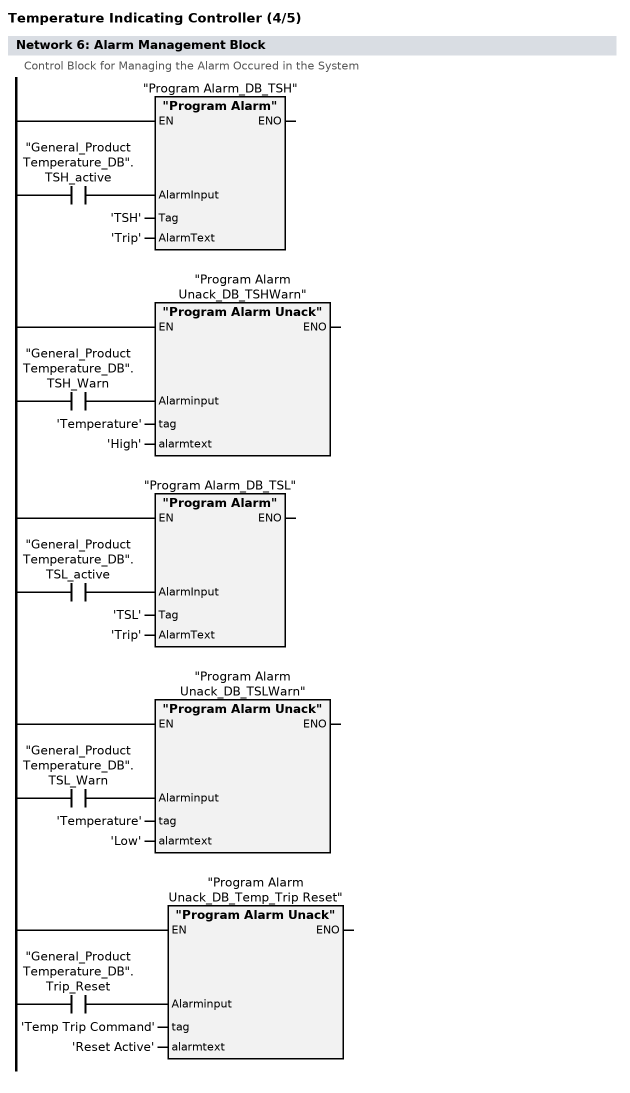
   RUNG wire#powerrail
      "Program Alarm_DB_TSH"(AlarmInput := wire#w1, Tag := 'TSH', AlarmText := 'Trip')
   END_RUNG
   RUNG wire#powerrail
      Contact( "General_Product Temperature_DB".TSH_active )
   END_RUNG wire#w1
   RUNG wire#powerrail
      "Program Alarm Unack_DB_TSHWarn"(Alarminput := wire#w2, tag := 'Temperature', alarmtext := 'High')
   END_RUNG
   RUNG wire#powerrail
      Contact( "General_Product Temperature_DB".TSH_Warn )
   END_RUNG wire#w2
   RUNG wire#powerrail
      "Program Alarm_DB_TSL"(AlarmInput := wire#w3, Tag := 'TSL', AlarmText := 'Trip')
   END_RUNG
   RUNG wire#powerrail
      Contact( "General_Product Temperature_DB".TSL_active )
   END_RUNG wire#w3
   RUNG wire#powerrail
      "Program Alarm Unack_DB_TSLWarn"(Alarminput := wire#w4, tag := 'Temperature', alarmtext := 'Low')
   END_RUNG
   RUNG wire#powerrail
      Contact( "General_Product Temperature_DB".TSL_Warn )
   END_RUNG wire#w4
   RUNG wire#powerrail
      "Program Alarm Unack_DB_Temp_Trip Reset"(Alarminput := wire#w5, tag := 'Temp Trip Command', alarmtext := 'Reset Active')
   END_RUNG
   RUNG wire#powerrail
      Contact( "General_Product Temperature_DB".Trip_Reset )
   END_RUNG wire#w5
   // the same network as SCL:
   "Program Alarm_DB_TSH"(AlarmInput := "General_Product Temperature_DB".TSH_active,   // "Program Alarm"
                          Tag := 'TSH',
                          AlarmText := 'Trip');
   "Program Alarm Unack_DB_TSHWarn"(Alarminput := "General_Product Temperature_DB".TSH_Warn,   // "Program Alarm Unack"
                           tag := 'Temperature',
                           alarmtext := 'High');
   "Program Alarm_DB_TSL"(AlarmInput := "General_Product Temperature_DB".TSL_active,   // "Program Alarm"
                          Tag := 'TSL',
                          AlarmText := 'Trip');
   "Program Alarm Unack_DB_TSLWarn"(Alarminput := "General_Product Temperature_DB".TSL_Warn,   // "Program Alarm Unack"
                           tag := 'Temperature',
                           alarmtext := 'Low');
   "Program Alarm Unack_DB_Temp_Trip Reset"(Alarminput := "General_Product Temperature_DB".Trip_Reset,   // "Program Alarm Unack"
                           tag := 'Temp Trip Command',
                           alarmtext := 'Reset Active');
END_REGION

REGION Network 7: User Additional Feature
   // Put additional feature that user can use to easier the system operation
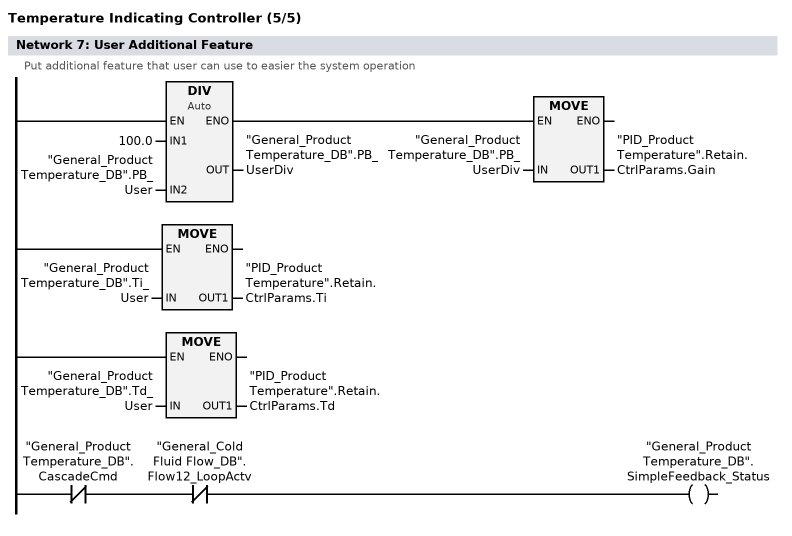
   RUNG wire#powerrail
      Div(in1 := 100.0, in2 := "General_Product Temperature_DB".PB_User, out => "General_Product Temperature_DB".PB_UserDiv)
      Move(in := "General_Product Temperature_DB".PB_UserDiv, out1 => "PID_Product Temperature".Retain.CtrlParams.Gain)
   END_RUNG
   RUNG wire#powerrail
      Move(in := "General_Product Temperature_DB".Ti_User, out1 => "PID_Product Temperature".Retain.CtrlParams.Ti)
   END_RUNG
   RUNG wire#powerrail
      Move(in := "General_Product Temperature_DB".Td_User, out1 => "PID_Product Temperature".Retain.CtrlParams.Td)
   END_RUNG
   RUNG wire#powerrail
      I_Contact( "General_Product Temperature_DB".CascadeCmd )
      I_Contact( "General_Cold Fluid Flow_DB".Flow12_LoopActv )
      Coil( "General_Product Temperature_DB".SimpleFeedback_Status )
   END_RUNG
   // the same network as SCL:
   "General_Product Temperature_DB".PB_UserDiv := 100.0 / "General_Product Temperature_DB".PB_User;
   "PID_Product Temperature".Retain.CtrlParams.Gain := "General_Product Temperature_DB".PB_UserDiv;
   "PID_Product Temperature".Retain.CtrlParams.Ti := "General_Product Temperature_DB".Ti_User;
   "PID_Product Temperature".Retain.CtrlParams.Td := "General_Product Temperature_DB".Td_User;
   "General_Product Temperature_DB".SimpleFeedback_Status := NOT "General_Product Temperature_DB".CascadeCmd AND NOT "General_Cold Fluid Flow_DB".Flow12_LoopActv;
END_REGION
END_ORGANIZATION_BLOCK

ORGANIZATION_BLOCK "Flow Indicating Controller 11"   // OB33, LAD, CyclicInterrupt
TITLE = Flow Indicator Controller 11 (Hot Fluid)
{ S7_Optimized_Access := 'TRUE' }
VERSION : 0.1
// Ladder and Block Program to control flowrate of Hot Fluid (Tank Input)
   VAR_INPUT
      Initial_Call : Bool;   // Initial call of this OB
      Event_Count : Int;   // Events discarded
   END_VAR
BEGIN

REGION Network 1: User Setpoint
   // User input their Setpoint for flowrate in L/s  converted into Real Number for PID Setpoint (0-100)
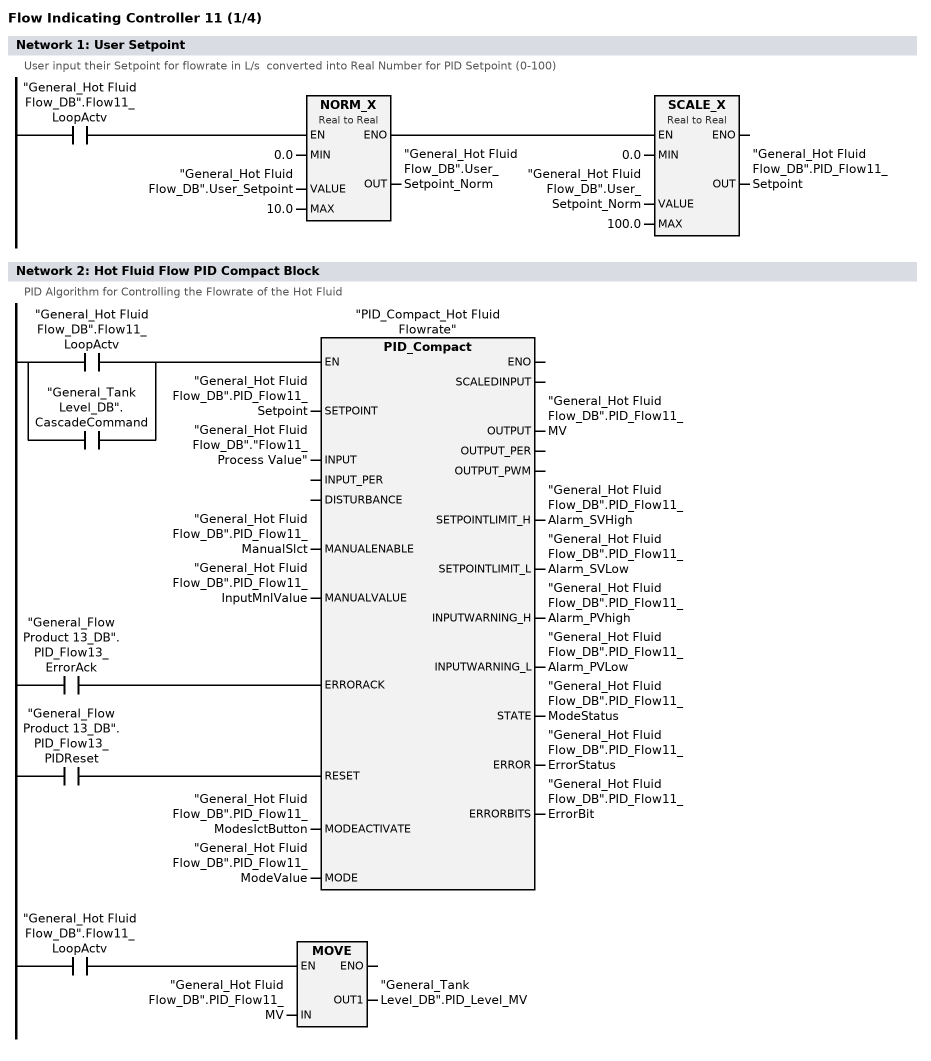
   RUNG wire#powerrail
      Contact( "General_Hot Fluid Flow_DB".Flow11_LoopActv )
      { S7_Templates := "[SrcType := Real, DestType := Real]" } Normalize(min := 0.0, value := "General_Hot Fluid Flow_DB".User_Setpoint, max := 10.0, out => "General_Hot Fluid Flow_DB".User_Setpoint_Norm)
      { S7_Templates := "[SrcType := Real, DestType := Real]" } Scale(min := 0.0, value := "General_Hot Fluid Flow_DB".User_Setpoint_Norm, max := 100.0, out => "General_Hot Fluid Flow_DB".PID_Flow11_Setpoint)
   END_RUNG
   // the same network as SCL:
   IF "General_Hot Fluid Flow_DB".Flow11_LoopActv THEN
       "General_Hot Fluid Flow_DB".User_Setpoint_Norm := NORM_X(MIN := 0.0, VALUE := "General_Hot Fluid Flow_DB".User_Setpoint, MAX := 10.0);
       "General_Hot Fluid Flow_DB".PID_Flow11_Setpoint := SCALE_X(MIN := 0.0, VALUE := "General_Hot Fluid Flow_DB".User_Setpoint_Norm, MAX := 100.0);
   END_IF;
END_REGION

REGION Network 2: Hot Fluid Flow PID Compact Block
   // PID Algorithm for Controlling the Flowrate of the Hot Fluid
   IF "General_Hot Fluid Flow_DB".Flow11_LoopActv OR "General_Tank Level_DB".CascadeCommand THEN
       "PID_Compact_Hot Fluid Flowrate"(Setpoint := "General_Hot Fluid Flow_DB".PID_Flow11_Setpoint,   // PID_Compact
                               Input := "General_Hot Fluid Flow_DB"."Flow11_Process Value",
                               ManualEnable := "General_Hot Fluid Flow_DB".PID_Flow11_ManualSlct,
                               ManualValue := "General_Hot Fluid Flow_DB".PID_Flow11_InputMnlValue,
                               ErrorAck := "General_Flow Product 13_DB".PID_Flow13_ErrorAck,
                               Reset := "General_Flow Product 13_DB".PID_Flow13_PIDReset,
                               ModeActivate := "General_Hot Fluid Flow_DB".PID_Flow11_ModeslctButton,
                               Mode := "General_Hot Fluid Flow_DB".PID_Flow11_ModeValue,
                               Output => "General_Hot Fluid Flow_DB".PID_Flow11_MV,
                               SetpointLimit_H => "General_Hot Fluid Flow_DB".PID_Flow11_Alarm_SVHigh,
                               SetpointLimit_L => "General_Hot Fluid Flow_DB".PID_Flow11_Alarm_SVLow,
                               InputWarning_H => "General_Hot Fluid Flow_DB".PID_Flow11_Alarm_PVhigh,
                               InputWarning_L => "General_Hot Fluid Flow_DB".PID_Flow11_Alarm_PVLow,
                               State => "General_Hot Fluid Flow_DB".PID_Flow11_ModeStatus,
                               Error => "General_Hot Fluid Flow_DB".PID_Flow11_ErrorStatus,
                               ErrorBits => "General_Hot Fluid Flow_DB".PID_Flow11_ErrorBit);
   END_IF;
   IF "General_Hot Fluid Flow_DB".Flow11_LoopActv THEN
       "General_Tank Level_DB".PID_Level_MV := "General_Hot Fluid Flow_DB".PID_Flow11_MV;
   END_IF;
END_REGION

REGION Network 3: Hot Fluid Process Control Block
   // Process for Flowrate as First Order System
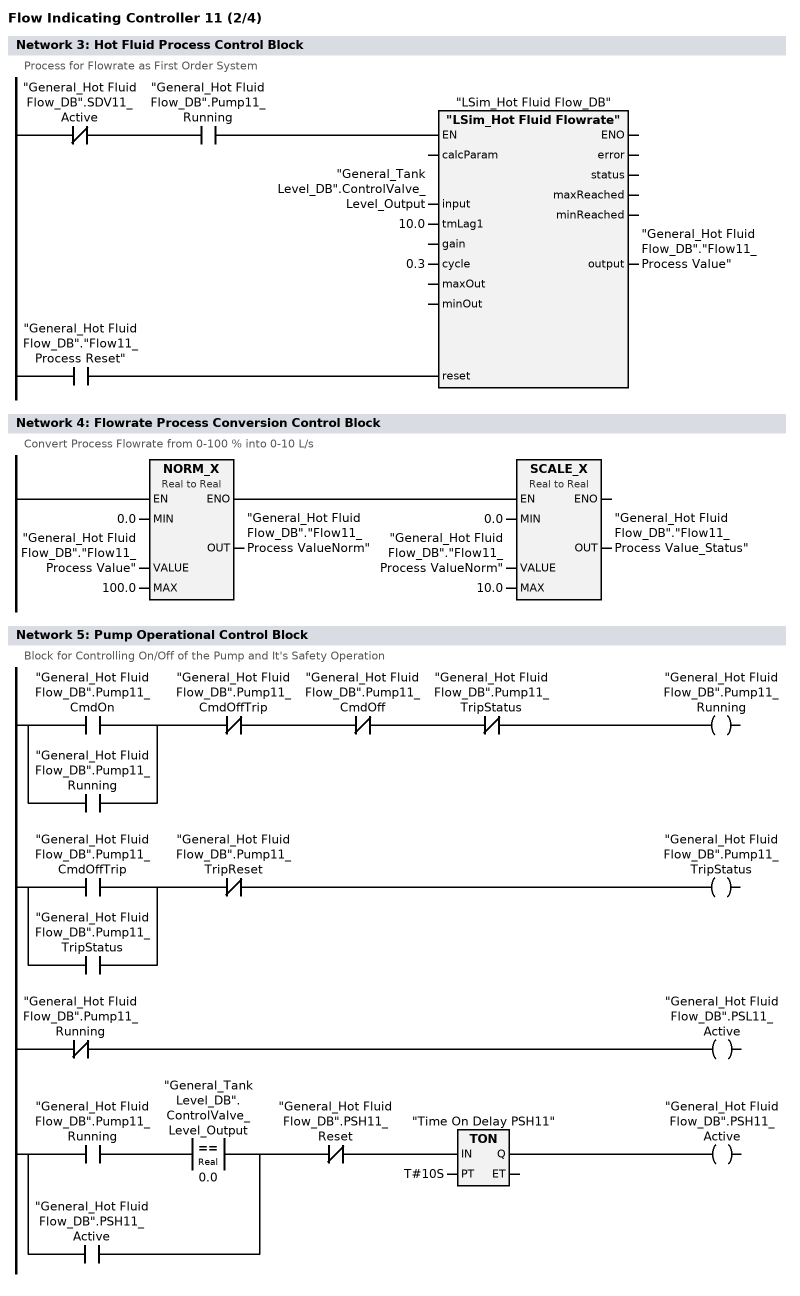
   RUNG wire#powerrail
      I_Contact( "General_Hot Fluid Flow_DB".SDV11_Active )
      Contact( "General_Hot Fluid Flow_DB".Pump11_Running )
      "LSim_Hot Fluid Flow_DB"(reset := wire#w1, calcParam :=, input := "General_Tank Level_DB".ControlValve_Level_Output, tmLag1 := 10.0, gain :=, cycle := 0.3, maxOut :=, minOut :=, error =>, status =>, maxReached =>, minReached =>, output => "General_Hot Fluid Flow_DB"."Flow11_Process Value")
   END_RUNG
   RUNG wire#powerrail
      Contact( "General_Hot Fluid Flow_DB"."Flow11_Process Reset" )
   END_RUNG wire#w1
   // the same network as SCL:
   IF NOT "General_Hot Fluid Flow_DB".SDV11_Active AND "General_Hot Fluid Flow_DB".Pump11_Running THEN
       "LSim_Hot Fluid Flow_DB"(input := "General_Tank Level_DB".ControlValve_Level_Output,   // "LSim_Hot Fluid Flowrate"
                               tmLag1 := 10.0,
                               cycle := 0.3,
                               reset := "General_Hot Fluid Flow_DB"."Flow11_Process Reset",
                               output => "General_Hot Fluid Flow_DB"."Flow11_Process Value");
   END_IF;
END_REGION

REGION Network 4: Flowrate Process Conversion Control Block
   // Convert Process Flowrate from 0-100 % into 0-10 L/s
   RUNG wire#powerrail
      { S7_Templates := "[SrcType := Real, DestType := Real]" } Normalize(min := 0.0, value := "General_Hot Fluid Flow_DB"."Flow11_Process Value", max := 100.0, out => "General_Hot Fluid Flow_DB"."Flow11_Process ValueNorm")
      { S7_Templates := "[SrcType := Real, DestType := Real]" } Scale(min := 0.0, value := "General_Hot Fluid Flow_DB"."Flow11_Process ValueNorm", max := 10.0, out => "General_Hot Fluid Flow_DB"."Flow11_Process Value_Status")
   END_RUNG
   // the same network as SCL:
   "General_Hot Fluid Flow_DB"."Flow11_Process ValueNorm" := NORM_X(MIN := 0.0, VALUE := "General_Hot Fluid Flow_DB"."Flow11_Process Value", MAX := 100.0);
   "General_Hot Fluid Flow_DB"."Flow11_Process Value_Status" := SCALE_X(MIN := 0.0, VALUE := "General_Hot Fluid Flow_DB"."Flow11_Process ValueNorm", MAX := 10.0);
END_REGION

REGION Network 5: Pump Operational Control Block
   // Block for Controlling On/Off of the Pump and It's Safety Operation
   "General_Hot Fluid Flow_DB".Pump11_Running := ("General_Hot Fluid Flow_DB".Pump11_CmdOn OR "General_Hot Fluid Flow_DB".Pump11_Running) AND NOT "General_Hot Fluid Flow_DB".Pump11_CmdOffTrip AND NOT "General_Hot Fluid Flow_DB".Pump11_CmdOff AND NOT "General_Hot Fluid Flow_DB".Pump11_TripStatus;
   "General_Hot Fluid Flow_DB".Pump11_TripStatus := ("General_Hot Fluid Flow_DB".Pump11_CmdOffTrip OR "General_Hot Fluid Flow_DB".Pump11_TripStatus) AND NOT "General_Hot Fluid Flow_DB".Pump11_TripReset;
   "General_Hot Fluid Flow_DB".PSL11_Active := NOT "General_Hot Fluid Flow_DB".Pump11_Running;
   "Time On Delay PSH11".TON(IN := (("General_Hot Fluid Flow_DB".Pump11_Running AND ("General_Tank Level_DB".ControlValve_Level_Output = 0.0)) OR "General_Hot Fluid Flow_DB".PSH11_Active) AND NOT "General_Hot Fluid Flow_DB".PSH11_Reset,
                           PT := T#10S);
   "General_Hot Fluid Flow_DB".PSH11_Active := "Time On Delay PSH11".Q;
END_REGION

REGION Network 6: Alarm Management Block
   // Control Block for Managing the Alarm Occured in the System
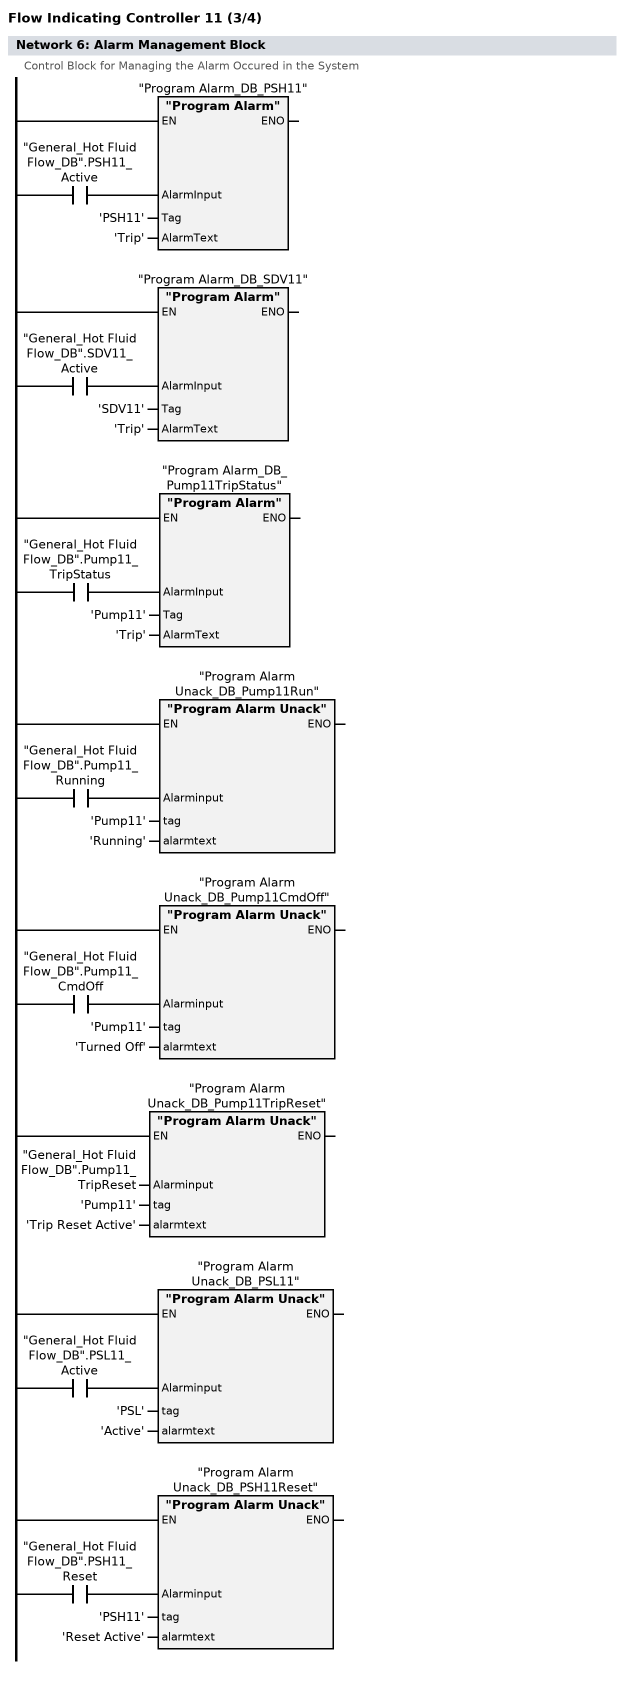
   RUNG wire#powerrail
      "Program Alarm_DB_PSH11"(AlarmInput := wire#w1, Tag := 'PSH11', AlarmText := 'Trip')
   END_RUNG
   RUNG wire#powerrail
      Contact( "General_Hot Fluid Flow_DB".PSH11_Active )
   END_RUNG wire#w1
   RUNG wire#powerrail
      "Program Alarm_DB_SDV11"(AlarmInput := wire#w2, Tag := 'SDV11', AlarmText := 'Trip')
   END_RUNG
   RUNG wire#powerrail
      Contact( "General_Hot Fluid Flow_DB".SDV11_Active )
   END_RUNG wire#w2
   RUNG wire#powerrail
      "Program Alarm_DB_Pump11TripStatus"(AlarmInput := wire#w3, Tag := 'Pump11', AlarmText := 'Trip')
   END_RUNG
   RUNG wire#powerrail
      Contact( "General_Hot Fluid Flow_DB".Pump11_TripStatus )
   END_RUNG wire#w3
   RUNG wire#powerrail
      "Program Alarm Unack_DB_Pump11Run"(Alarminput := wire#w4, tag := 'Pump11', alarmtext := 'Running')
   END_RUNG
   RUNG wire#powerrail
      Contact( "General_Hot Fluid Flow_DB".Pump11_Running )
   END_RUNG wire#w4
   RUNG wire#powerrail
      "Program Alarm Unack_DB_Pump11CmdOff"(Alarminput := wire#w5, tag := 'Pump11', alarmtext := 'Turned Off')
   END_RUNG
   RUNG wire#powerrail
      Contact( "General_Hot Fluid Flow_DB".Pump11_CmdOff )
   END_RUNG wire#w5
   RUNG wire#powerrail
      "Program Alarm Unack_DB_Pump11TripReset"(Alarminput := "General_Hot Fluid Flow_DB".Pump11_TripReset, tag := 'Pump11', alarmtext := 'Trip Reset Active')
   END_RUNG
   RUNG wire#powerrail
      "Program Alarm Unack_DB_PSL11"(Alarminput := wire#w6, tag := 'PSL', alarmtext := 'Active')
   END_RUNG
   RUNG wire#powerrail
      Contact( "General_Hot Fluid Flow_DB".PSL11_Active )
   END_RUNG wire#w6
   RUNG wire#powerrail
      "Program Alarm Unack_DB_PSH11Reset"(Alarminput := wire#w7, tag := 'PSH11', alarmtext := 'Reset Active')
   END_RUNG
   RUNG wire#powerrail
      Contact( "General_Hot Fluid Flow_DB".PSH11_Reset )
   END_RUNG wire#w7
   // the same network as SCL:
   "Program Alarm_DB_PSH11"(AlarmInput := "General_Hot Fluid Flow_DB".PSH11_Active,   // "Program Alarm"
                           Tag := 'PSH11',
                           AlarmText := 'Trip');
   "Program Alarm_DB_SDV11"(AlarmInput := "General_Hot Fluid Flow_DB".SDV11_Active,   // "Program Alarm"
                           Tag := 'SDV11',
                           AlarmText := 'Trip');
   "Program Alarm_DB_Pump11TripStatus"(AlarmInput := "General_Hot Fluid Flow_DB".Pump11_TripStatus,   // "Program Alarm"
                           Tag := 'Pump11',
                           AlarmText := 'Trip');
   "Program Alarm Unack_DB_Pump11Run"(Alarminput := "General_Hot Fluid Flow_DB".Pump11_Running,   // "Program Alarm Unack"
                           tag := 'Pump11',
                           alarmtext := 'Running');
   "Program Alarm Unack_DB_Pump11CmdOff"(Alarminput := "General_Hot Fluid Flow_DB".Pump11_CmdOff,   // "Program Alarm Unack"
                           tag := 'Pump11',
                           alarmtext := 'Turned Off');
   "Program Alarm Unack_DB_Pump11TripReset"(Alarminput := "General_Hot Fluid Flow_DB".Pump11_TripReset,   // "Program Alarm Unack"
                           tag := 'Pump11',
                           alarmtext := 'Trip Reset Active');
   "Program Alarm Unack_DB_PSL11"(Alarminput := "General_Hot Fluid Flow_DB".PSL11_Active,   // "Program Alarm Unack"
                           tag := 'PSL',
                           alarmtext := 'Active');
   "Program Alarm Unack_DB_PSH11Reset"(Alarminput := "General_Hot Fluid Flow_DB".PSH11_Reset,   // "Program Alarm Unack"
                           tag := 'PSH11',
                           alarmtext := 'Reset Active');
END_REGION

REGION Network 7: User Additional Feature
   // Put additional feature that user can use to easier the system operation
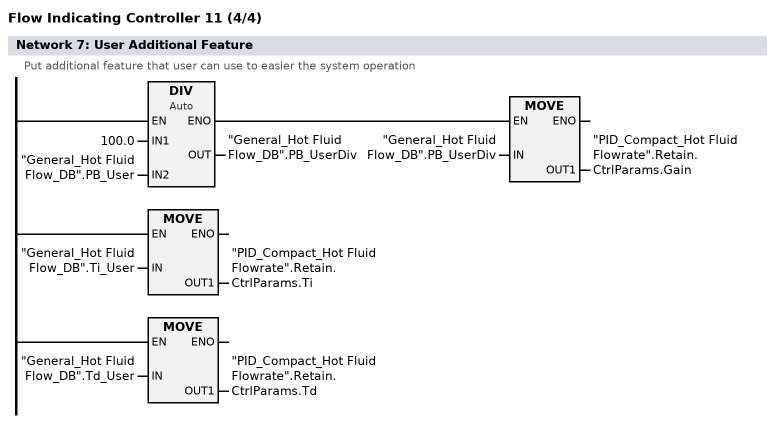
   RUNG wire#powerrail
      Div(in1 := 100.0, in2 := "General_Hot Fluid Flow_DB".PB_User, out => "General_Hot Fluid Flow_DB".PB_UserDiv)
      Move(in := "General_Hot Fluid Flow_DB".PB_UserDiv, out1 => "PID_Compact_Hot Fluid Flowrate".Retain.CtrlParams.Gain)
   END_RUNG
   RUNG wire#powerrail
      Move(in := "General_Hot Fluid Flow_DB".Ti_User, out1 => "PID_Compact_Hot Fluid Flowrate".Retain.CtrlParams.Ti)
   END_RUNG
   RUNG wire#powerrail
      Move(in := "General_Hot Fluid Flow_DB".Td_User, out1 => "PID_Compact_Hot Fluid Flowrate".Retain.CtrlParams.Td)
   END_RUNG
   // the same network as SCL:
   "General_Hot Fluid Flow_DB".PB_UserDiv := 100.0 / "General_Hot Fluid Flow_DB".PB_User;
   "PID_Compact_Hot Fluid Flowrate".Retain.CtrlParams.Gain := "General_Hot Fluid Flow_DB".PB_UserDiv;
   "PID_Compact_Hot Fluid Flowrate".Retain.CtrlParams.Ti := "General_Hot Fluid Flow_DB".Ti_User;
   "PID_Compact_Hot Fluid Flowrate".Retain.CtrlParams.Td := "General_Hot Fluid Flow_DB".Td_User;
END_REGION
END_ORGANIZATION_BLOCK

ORGANIZATION_BLOCK "Flow Indicating Controller 12"   // OB34, LAD, CyclicInterrupt
TITLE = Flow Indicator Controller 12 (Cold Fluid)
{ S7_Optimized_Access := 'TRUE' }
VERSION : 0.1
// Ladder and Block Program to control flowrate of Cold Fluid (Tank Input)
   VAR_INPUT
      Initial_Call : Bool;   // Initial call of this OB
      Event_Count : Int;   // Events discarded
   END_VAR
BEGIN

REGION Network 1: User Setpoint
   // User input their Setpoint for flowrate in L/s  converted into Real Number for PID Setpoint (0-100)
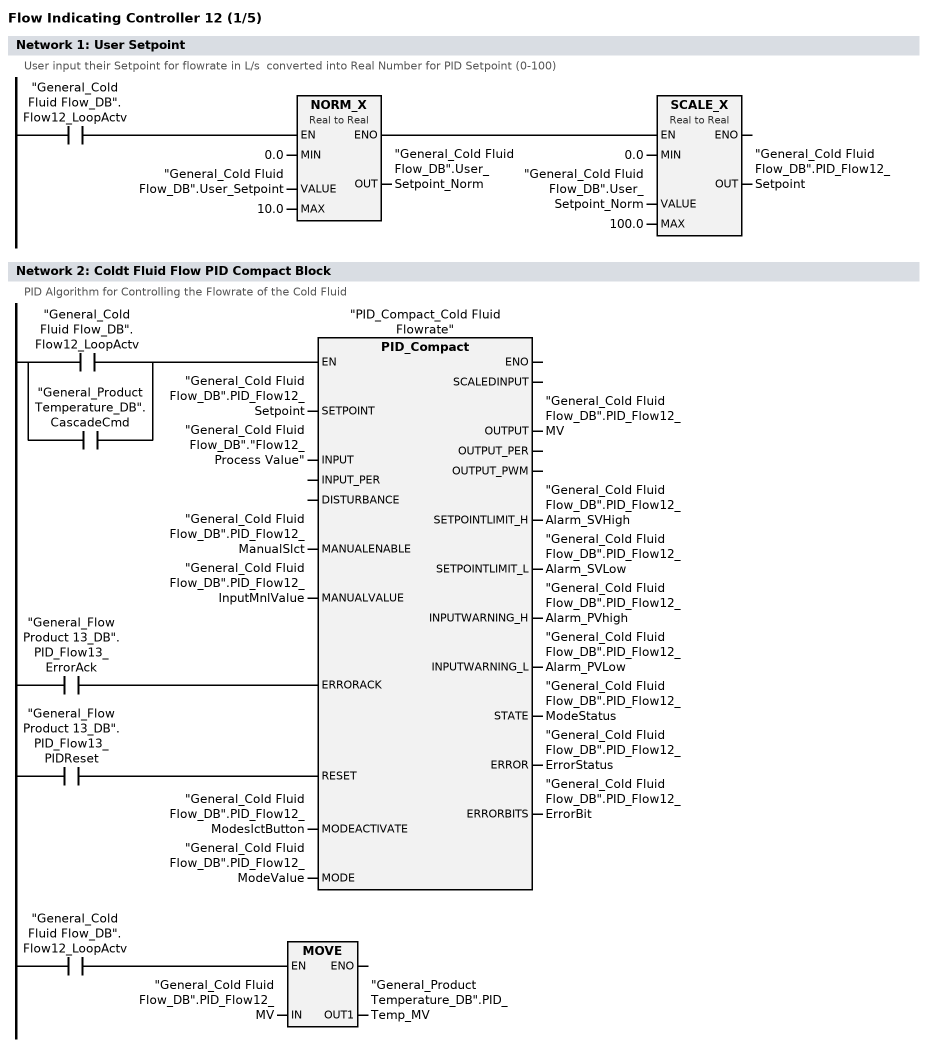
   RUNG wire#powerrail
      Contact( "General_Cold Fluid Flow_DB".Flow12_LoopActv )
      { S7_Templates := "[SrcType := Real, DestType := Real]" } Normalize(min := 0.0, value := "General_Cold Fluid Flow_DB".User_Setpoint, max := 10.0, out => "General_Cold Fluid Flow_DB".User_Setpoint_Norm)
      { S7_Templates := "[SrcType := Real, DestType := Real]" } Scale(min := 0.0, value := "General_Cold Fluid Flow_DB".User_Setpoint_Norm, max := 100.0, out => "General_Cold Fluid Flow_DB".PID_Flow12_Setpoint)
   END_RUNG
   // the same network as SCL:
   IF "General_Cold Fluid Flow_DB".Flow12_LoopActv THEN
       "General_Cold Fluid Flow_DB".User_Setpoint_Norm := NORM_X(MIN := 0.0, VALUE := "General_Cold Fluid Flow_DB".User_Setpoint, MAX := 10.0);
       "General_Cold Fluid Flow_DB".PID_Flow12_Setpoint := SCALE_X(MIN := 0.0, VALUE := "General_Cold Fluid Flow_DB".User_Setpoint_Norm, MAX := 100.0);
   END_IF;
END_REGION

REGION Network 2: Coldt Fluid Flow PID Compact Block
   // PID Algorithm for Controlling the Flowrate of the Cold Fluid
   IF "General_Cold Fluid Flow_DB".Flow12_LoopActv OR "General_Product Temperature_DB".CascadeCmd THEN
       "PID_Compact_Cold Fluid Flowrate"(Setpoint := "General_Cold Fluid Flow_DB".PID_Flow12_Setpoint,   // PID_Compact
                               Input := "General_Cold Fluid Flow_DB"."Flow12_Process Value",
                               ManualEnable := "General_Cold Fluid Flow_DB".PID_Flow12_ManualSlct,
                               ManualValue := "General_Cold Fluid Flow_DB".PID_Flow12_InputMnlValue,
                               ErrorAck := "General_Flow Product 13_DB".PID_Flow13_ErrorAck,
                               Reset := "General_Flow Product 13_DB".PID_Flow13_PIDReset,
                               ModeActivate := "General_Cold Fluid Flow_DB".PID_Flow12_ModeslctButton,
                               Mode := "General_Cold Fluid Flow_DB".PID_Flow12_ModeValue,
                               Output => "General_Cold Fluid Flow_DB".PID_Flow12_MV,
                               SetpointLimit_H => "General_Cold Fluid Flow_DB".PID_Flow12_Alarm_SVHigh,
                               SetpointLimit_L => "General_Cold Fluid Flow_DB".PID_Flow12_Alarm_SVLow,
                               InputWarning_H => "General_Cold Fluid Flow_DB".PID_Flow12_Alarm_PVhigh,
                               InputWarning_L => "General_Cold Fluid Flow_DB".PID_Flow12_Alarm_PVLow,
                               State => "General_Cold Fluid Flow_DB".PID_Flow12_ModeStatus,
                               Error => "General_Cold Fluid Flow_DB".PID_Flow12_ErrorStatus,
                               ErrorBits => "General_Cold Fluid Flow_DB".PID_Flow12_ErrorBit);
   END_IF;
   IF "General_Cold Fluid Flow_DB".Flow12_LoopActv THEN
       "General_Product Temperature_DB".PID_Temp_MV := "General_Cold Fluid Flow_DB".PID_Flow12_MV;
   END_IF;
END_REGION

REGION Network 3: Cold Fluid Process Control Block
   // Process for Flowrate as First Order System
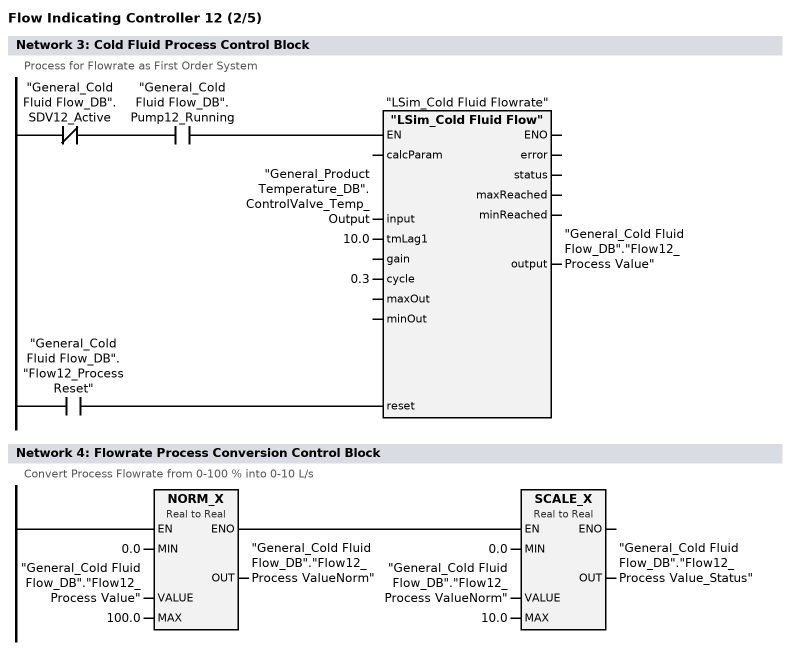
   RUNG wire#powerrail
      I_Contact( "General_Cold Fluid Flow_DB".SDV12_Active )
      Contact( "General_Cold Fluid Flow_DB".Pump12_Running )
      "LSim_Cold Fluid Flowrate"(reset := wire#w1, calcParam :=, input := "General_Product Temperature_DB".ControlValve_Temp_Output, tmLag1 := 10.0, gain :=, cycle := 0.3, maxOut :=, minOut :=, error =>, status =>, maxReached =>, minReached =>, output => "General_Cold Fluid Flow_DB"."Flow12_Process Value")
   END_RUNG
   RUNG wire#powerrail
      Contact( "General_Cold Fluid Flow_DB"."Flow12_Process Reset" )
   END_RUNG wire#w1
   // the same network as SCL:
   IF NOT "General_Cold Fluid Flow_DB".SDV12_Active AND "General_Cold Fluid Flow_DB".Pump12_Running THEN
       "LSim_Cold Fluid Flowrate"(input := "General_Product Temperature_DB".ControlValve_Temp_Output,   // "LSim_Cold Fluid Flow"
                               tmLag1 := 10.0,
                               cycle := 0.3,
                               reset := "General_Cold Fluid Flow_DB"."Flow12_Process Reset",
                               output => "General_Cold Fluid Flow_DB"."Flow12_Process Value");
   END_IF;
END_REGION

REGION Network 4: Flowrate Process Conversion Control Block
   // Convert Process Flowrate from 0-100 % into 0-10 L/s
   RUNG wire#powerrail
      { S7_Templates := "[SrcType := Real, DestType := Real]" } Normalize(min := 0.0, value := "General_Cold Fluid Flow_DB"."Flow12_Process Value", max := 100.0, out => "General_Cold Fluid Flow_DB"."Flow12_Process ValueNorm")
      { S7_Templates := "[SrcType := Real, DestType := Real]" } Scale(min := 0.0, value := "General_Cold Fluid Flow_DB"."Flow12_Process ValueNorm", max := 10.0, out => "General_Cold Fluid Flow_DB"."Flow12_Process Value_Status")
   END_RUNG
   // the same network as SCL:
   "General_Cold Fluid Flow_DB"."Flow12_Process ValueNorm" := NORM_X(MIN := 0.0, VALUE := "General_Cold Fluid Flow_DB"."Flow12_Process Value", MAX := 100.0);
   "General_Cold Fluid Flow_DB"."Flow12_Process Value_Status" := SCALE_X(MIN := 0.0, VALUE := "General_Cold Fluid Flow_DB"."Flow12_Process ValueNorm", MAX := 10.0);
END_REGION

REGION Network 5: Pump Operational Control Block
   // Block for Controlling On/Off of the Pump and It's Safety Operation
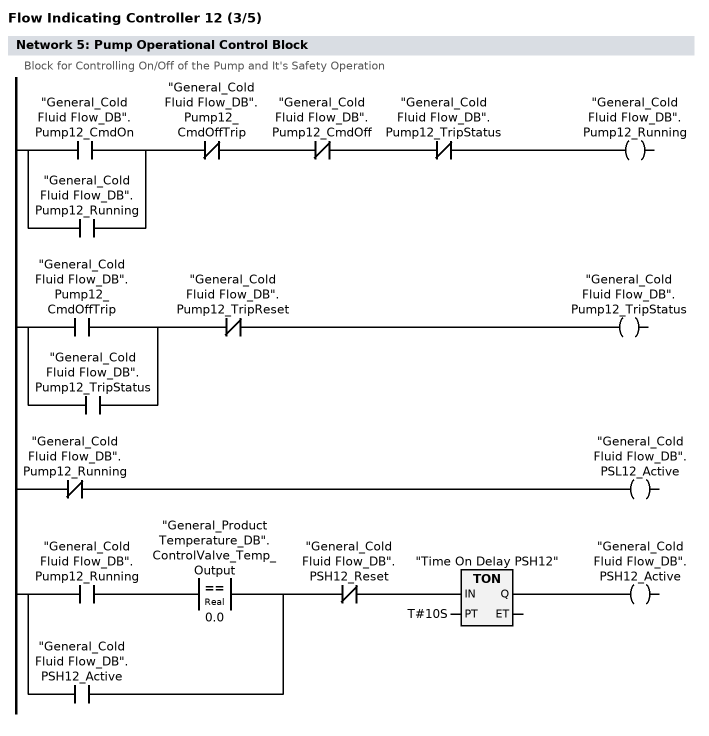
   "General_Cold Fluid Flow_DB".Pump12_Running := ("General_Cold Fluid Flow_DB".Pump12_CmdOn OR "General_Cold Fluid Flow_DB".Pump12_Running) AND NOT "General_Cold Fluid Flow_DB".Pump12_CmdOffTrip AND NOT "General_Cold Fluid Flow_DB".Pump12_CmdOff AND NOT "General_Cold Fluid Flow_DB".Pump12_TripStatus;
   "General_Cold Fluid Flow_DB".Pump12_TripStatus := ("General_Cold Fluid Flow_DB".Pump12_CmdOffTrip OR "General_Cold Fluid Flow_DB".Pump12_TripStatus) AND NOT "General_Cold Fluid Flow_DB".Pump12_TripReset;
   "General_Cold Fluid Flow_DB".PSL12_Active := NOT "General_Cold Fluid Flow_DB".Pump12_Running;
   "Time On Delay PSH12".TON(IN := (("General_Cold Fluid Flow_DB".Pump12_Running AND ("General_Product Temperature_DB".ControlValve_Temp_Output = 0.0)) OR "General_Cold Fluid Flow_DB".PSH12_Active) AND NOT "General_Cold Fluid Flow_DB".PSH12_Reset,
                           PT := T#10S);
   "General_Cold Fluid Flow_DB".PSH12_Active := "Time On Delay PSH12".Q;
END_REGION

REGION Network 6: Alarm Management Block
   // Control Block for Managing the Alarm Occured in the System
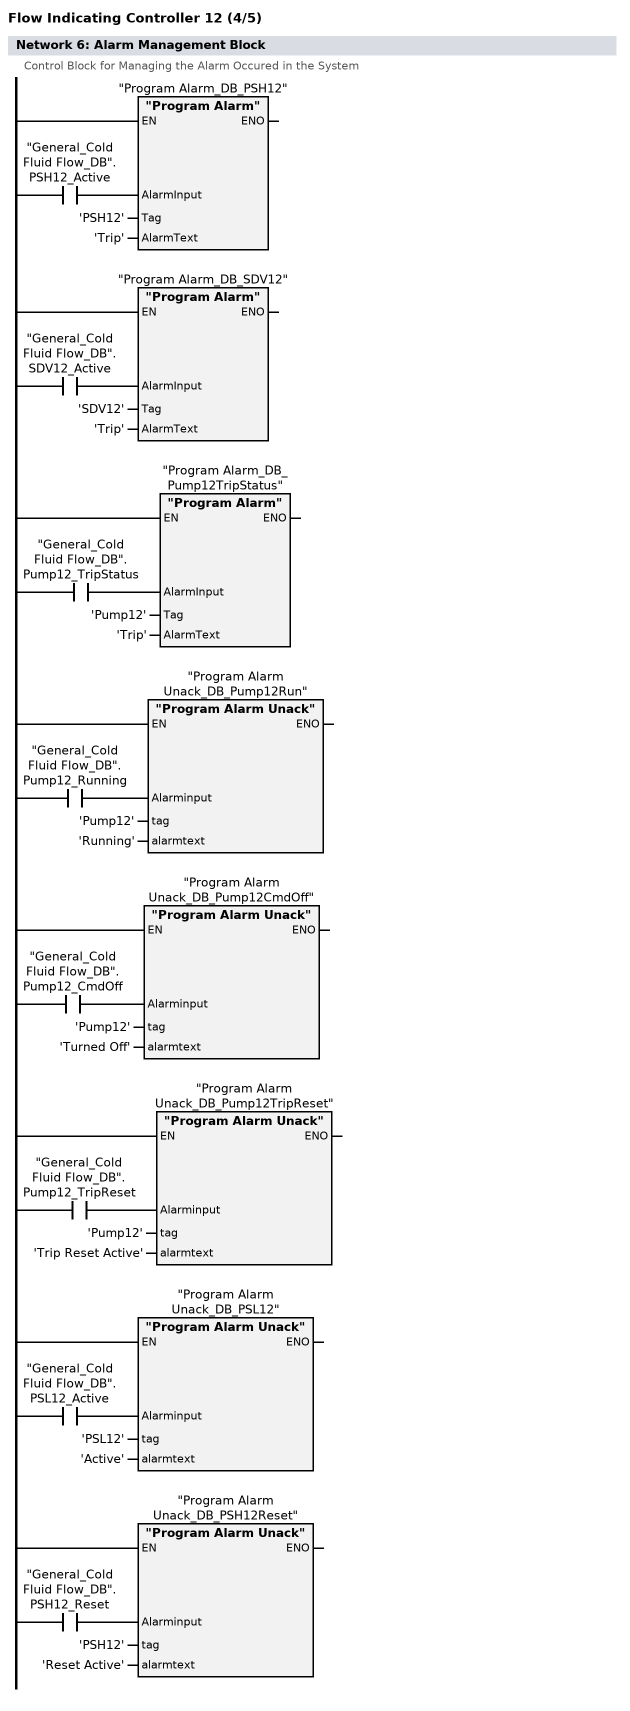
   RUNG wire#powerrail
      "Program Alarm_DB_PSH12"(AlarmInput := wire#w1, Tag := 'PSH12', AlarmText := 'Trip')
   END_RUNG
   RUNG wire#powerrail
      Contact( "General_Cold Fluid Flow_DB".PSH12_Active )
   END_RUNG wire#w1
   RUNG wire#powerrail
      "Program Alarm_DB_SDV12"(AlarmInput := wire#w2, Tag := 'SDV12', AlarmText := 'Trip')
   END_RUNG
   RUNG wire#powerrail
      Contact( "General_Cold Fluid Flow_DB".SDV12_Active )
   END_RUNG wire#w2
   RUNG wire#powerrail
      "Program Alarm_DB_Pump12TripStatus"(AlarmInput := wire#w3, Tag := 'Pump12', AlarmText := 'Trip')
   END_RUNG
   RUNG wire#powerrail
      Contact( "General_Cold Fluid Flow_DB".Pump12_TripStatus )
   END_RUNG wire#w3
   RUNG wire#powerrail
      "Program Alarm Unack_DB_Pump12Run"(Alarminput := wire#w4, tag := 'Pump12', alarmtext := 'Running')
   END_RUNG
   RUNG wire#powerrail
      Contact( "General_Cold Fluid Flow_DB".Pump12_Running )
   END_RUNG wire#w4
   RUNG wire#powerrail
      "Program Alarm Unack_DB_Pump12CmdOff"(Alarminput := wire#w5, tag := 'Pump12', alarmtext := 'Turned Off')
   END_RUNG
   RUNG wire#powerrail
      Contact( "General_Cold Fluid Flow_DB".Pump12_CmdOff )
   END_RUNG wire#w5
   RUNG wire#powerrail
      "Program Alarm Unack_DB_Pump12TripReset"(Alarminput := wire#w6, tag := 'Pump12', alarmtext := 'Trip Reset Active')
   END_RUNG
   RUNG wire#powerrail
      Contact( "General_Cold Fluid Flow_DB".Pump12_TripReset )
   END_RUNG wire#w6
   RUNG wire#powerrail
      "Program Alarm Unack_DB_PSL12"(Alarminput := wire#w7, tag := 'PSL12', alarmtext := 'Active')
   END_RUNG
   RUNG wire#powerrail
      Contact( "General_Cold Fluid Flow_DB".PSL12_Active )
   END_RUNG wire#w7
   RUNG wire#powerrail
      "Program Alarm Unack_DB_PSH12Reset"(Alarminput := wire#w8, tag := 'PSH12', alarmtext := 'Reset Active')
   END_RUNG
   RUNG wire#powerrail
      Contact( "General_Cold Fluid Flow_DB".PSH12_Reset )
   END_RUNG wire#w8
   // the same network as SCL:
   "Program Alarm_DB_PSH12"(AlarmInput := "General_Cold Fluid Flow_DB".PSH12_Active,   // "Program Alarm"
                           Tag := 'PSH12',
                           AlarmText := 'Trip');
   "Program Alarm_DB_SDV12"(AlarmInput := "General_Cold Fluid Flow_DB".SDV12_Active,   // "Program Alarm"
                           Tag := 'SDV12',
                           AlarmText := 'Trip');
   "Program Alarm_DB_Pump12TripStatus"(AlarmInput := "General_Cold Fluid Flow_DB".Pump12_TripStatus,   // "Program Alarm"
                           Tag := 'Pump12',
                           AlarmText := 'Trip');
   "Program Alarm Unack_DB_Pump12Run"(Alarminput := "General_Cold Fluid Flow_DB".Pump12_Running,   // "Program Alarm Unack"
                           tag := 'Pump12',
                           alarmtext := 'Running');
   "Program Alarm Unack_DB_Pump12CmdOff"(Alarminput := "General_Cold Fluid Flow_DB".Pump12_CmdOff,   // "Program Alarm Unack"
                           tag := 'Pump12',
                           alarmtext := 'Turned Off');
   "Program Alarm Unack_DB_Pump12TripReset"(Alarminput := "General_Cold Fluid Flow_DB".Pump12_TripReset,   // "Program Alarm Unack"
                           tag := 'Pump12',
                           alarmtext := 'Trip Reset Active');
   "Program Alarm Unack_DB_PSL12"(Alarminput := "General_Cold Fluid Flow_DB".PSL12_Active,   // "Program Alarm Unack"
                           tag := 'PSL12',
                           alarmtext := 'Active');
   "Program Alarm Unack_DB_PSH12Reset"(Alarminput := "General_Cold Fluid Flow_DB".PSH12_Reset,   // "Program Alarm Unack"
                           tag := 'PSH12',
                           alarmtext := 'Reset Active');
END_REGION

REGION Network 7: User Additional Feature
   // Put additional feature that user can use to easier the system operation
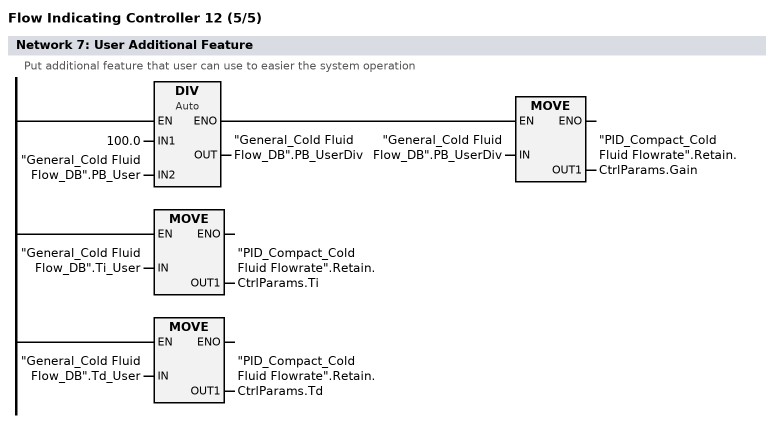
   RUNG wire#powerrail
      Div(in1 := 100.0, in2 := "General_Cold Fluid Flow_DB".PB_User, out => "General_Cold Fluid Flow_DB".PB_UserDiv)
      Move(in := "General_Cold Fluid Flow_DB".PB_UserDiv, out1 => "PID_Compact_Cold Fluid Flowrate".Retain.CtrlParams.Gain)
   END_RUNG
   RUNG wire#powerrail
      Move(in := "General_Cold Fluid Flow_DB".Ti_User, out1 => "PID_Compact_Cold Fluid Flowrate".Retain.CtrlParams.Ti)
   END_RUNG
   RUNG wire#powerrail
      Move(in := "General_Cold Fluid Flow_DB".Td_User, out1 => "PID_Compact_Cold Fluid Flowrate".Retain.CtrlParams.Td)
   END_RUNG
   // the same network as SCL:
   "General_Cold Fluid Flow_DB".PB_UserDiv := 100.0 / "General_Cold Fluid Flow_DB".PB_User;
   "PID_Compact_Cold Fluid Flowrate".Retain.CtrlParams.Gain := "General_Cold Fluid Flow_DB".PB_UserDiv;
   "PID_Compact_Cold Fluid Flowrate".Retain.CtrlParams.Ti := "General_Cold Fluid Flow_DB".Ti_User;
   "PID_Compact_Cold Fluid Flowrate".Retain.CtrlParams.Td := "General_Cold Fluid Flow_DB".Td_User;
END_REGION
END_ORGANIZATION_BLOCK